FUNCTION_BLOCK SawdustScale (* goFB_ignore *)
  (* Standard: 61499-2 *)
  (* Version 0.1, 2017-00-16, hpea485, UOA *)
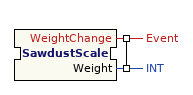
  EVENT_OUTPUT
    WeightChange WITH Weight;
  END_EVENT
  VAR_OUTPUT
    Weight : INT;
  END_VAR
  EC_STATES
    Start;
  END_STATES
END_FUNCTION_BLOCK
